TYPE E_CartJointState :
(
	CartJointState_Error := 1,
	CartJointState_Init := 2,
	CartJointState_SelfCheck := 3,
	CartJointState_Standby := 4,
	CartJointState_Ready := 5,
	CartJointState_InSurgery := 6,
	CartJointState_SteadyFootDeployment := 7,
	CartJointState_Movement := 8,
	CartJointState_HangAdjust := 9,
	CartJointState_AsepticDeployment := 10,
	CartJointState_RotaOverhang := 11,
	CartJointState_SlowStop := 12,
	
	CartJointState_totalNum := CartJointState_SlowStop
);
END_TYPE
//  CartJointState_totalNum = 'CartJointState_SlowStop'

(* stored: Version 1.1.0.1, ProductVersion 3.1.4024.12
   EnumerationTextList E_CartJointState: Id {6e3c6b3a-6c54-4485-8d03-0a28a138332d} *)
